PROGRAM MAIN
VAR
	iState 		: INT 	:= 0;	
	iMethod		: SINT 	:= 0;
	
	bCreateContainer	: 	BOOL := FALSE;
	bRemoveContainer	:	BOOL := FALSE;
	
	bSensorOben		: BOOL;
	bSensorMitte	: BOOL;
	bSensorUnten	: BOOL;
	bSensorLagerUnten		: BOOL;
	bSensorLagerMitte		: BOOL; 
	
	bHubmagnetOben	: BOOL := TRUE;
	bHubmagnetUnten	: BOOL := TRUE;
	
	
	
	instVereinzelung : Vereinzelung;
	counter : int := 0;
END_VAR

// Call models
instVereinzelung(
	ssMethodType:= iMethod, 
	Signal_CreateContainer:= BOOL_TO_LREAL(bCreateContainer), 
	c_Signal_RemoveContainerOnC:= bRemoveContainer, 
	SamplingTime:= 0.01, 
	Hw_HubmagnetOben:= bHubmagnetOben, 
	Hw_HubmagnetUnten:= bHubmagnetUnten, 
	Signal_Storage2=> bSensorLagerMitte, 
	Signal_Storage1=> bSensorLagerUnten, 
	Hw_SensorOben=> bSensorOben, 
	Hw_SensorMitte=> bSensorMitte, 
	Hw_SensorUnten=> bSensorUnten);


AdsVariables.Container1_ADS := BOOL_TO_REAL(bSensorUnten);
AdsVariables.Container2_ADS := BOOL_TO_REAL(bSensorMitte);
AdsVariables.Container3_ADS := BOOL_TO_REAL(bSensorOben);
AdsVariables.Container4_ADS := BOOL_TO_REAL(bSensorLagerUnten);
AdsVariables.Container5_ADS := BOOL_TO_REAL(bSensorLagerMitte);
AdsVariables.HubmagnetOben_ADS := BOOL_TO_REAL(bHubmagnetOben);
AdsVariables.HubmagnetUnten_ADS := BOOL_TO_REAL(bHubmagnetUnten);
	



// State Machine
CASE iState OF
	0:
		
		iState := iState +1;
	1:
		iMethod := 1;
END_CASE

END_PROGRAM

(* stored: Version 1.1.0.1, ProductVersion 3.1.4024.10
   POU MAIN: Id {fef2700b-e0b1-4384-91dc-030dd6cbb394}, SpecialFunc None *)
